Universal Robots PolyScope program: WIE2.urp

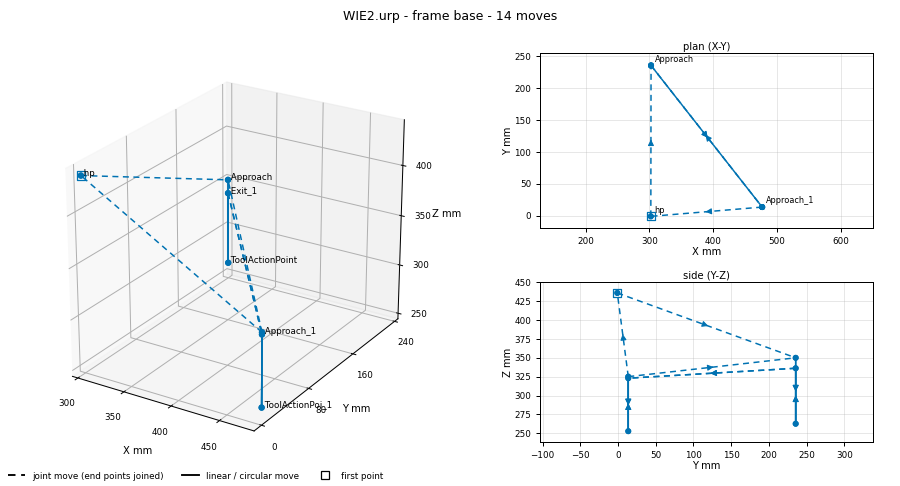
[picture p0: tool path of WIE2.urp in frame base, 14 of 14 moves have a stored position in this frame; points joined in program order, loops and branches not executed]
Program WIE2 (installation=default directory=/programs/Students createdIn=5.11.9.1010452 lastSavedIn=5.11.9.1010452 robotSerialNumber=20225200364)
Calibrated DH parameters: a=[0.00002, -0.569483, -0.54992, -0.00001, -0.000036, 0]; d=[0.180894, -146.691669, 192.918669, -46.053088, 0.119778, 0.115602]; alpha=[1.571425, -0.001534, 0.003359, 1.568739, -1.571477, 0]; deltaTheta=[0, 0.376258, -0.101074, -0.275185, -0.000002, 0]
Robot Program (runOnlyOnce=false)
  URCap RG Grip (OnRobot, OnRobot A/S) dataModel(rg-target-force=40.0, rg-target-width=0.1, Variable(key=on_return, variable(name=on_return)))
  MoveJ speed 60 deg/s, acceleration 80 deg/s^2 (useActiveTCP=true) feature=Base
    Waypoint hp: TCP in base x=302.217 y=-0.87 z=436.088 mm, rx=2.2254 ry=-2.21 rz=0.0041 rad; joints [35.141, -74.845, -127.965, -247.503, -90.009, -145.045] deg
    Loop Counting (count=3) loopVariable(name=Loop_1)
      URCap Palletizing (polyscope-pallet-impl, Universal Robots) dataModel(palletFeature=Base, isPalletizing=true, Variable(key=name, variable(name=Pallet_1)), Variable(key=globalCountingVariable, variable(name=Pallet_1_cnt_1, initializeExpression=1)), Variable(key=layerNumberVariable, variable(name=Pallet_1_lno, initializeExpression=1)), Variable(key=layerCountingVariable, variable(name=Pallet_1_lct, initializeExpression=1)), Variable(key=handleSeparatorVariable, variable(name=Pallet_1_sep, initializeExpression=False)), Variable(key=totalCountVariable, variable(name=Pallet_1_tct, initializeExpression=1)), Length(key=objectHeight value=0.00001 unit=M), Variable(key=referencePoint, variable(featureName=referencePoint)), Variable(key=separatorPoint, variable(featureName=separatorPoint))); state(isChildrenLocked=true)
        URCap Patterns (polyscope-pallet-impl, Universal Robots) state(isChildrenLocked=true)
          URCap Pattern (polyscope-pallet-impl, Universal Robots) dataModel(UUID=b11b03bd-8caf-4562-8920-b140e7a550b2, patternType=LINE, objects=3, Variable(key=nameVariable, variable(name=Line_Pattern_1))); state(isChildrenLocked=true)
            URCap Item (polyscope-pallet-impl, Universal Robots) dataModel(UUID=68741ad4-6990-4c8e-a16e-338bb588d268, patternType=LINE, index=0, calibrationDeltaTheta=[-2.1094217540068572E-7, 0.37625772532806073, -0.10107441100396769, -0.2751850025766889, -1.8024952768980196E-6, 2.9402326063437956E-8], calibrationA=[2.0416891277915125E-5, -0.5694828868469309, -0.5499202125525207, -9.504674691390763E-6, -3.603723657207661E-5, 0.0], calibrationD=[0.1808937726775539, -146.69166934821124, 192.91866861971778, -46.05308757405963, 0.11977780403821288, 0.11560212559305974], calibrationAlpha=[1.5714252480212174, -0.0015337665762078037, 0.0033588312559612306, 1.5687392298942362, -1.5714772428732047, 0.0], calibrationJointChecksum=[-1490546360, -1456574554, -1506622700, -1493399207, -1492840923, -1492940558], calibrationStatus=2, calibrationValidChecksum=true, baseToFeature=[0.0, 0.0, 0.0, 0.0, 0.0, 0.0], TCPOffset=[1.9606048756726224E-7, 3.440182682445947E-6, -6.058388327678799E-6, 3.4021623271823385E-5, 2.0407876993438444E-5, -5.7287062263560195E-5], Variable(key=variable, variable(name=StartItem_1)), JointPositions(key=jointpositions, JointPosition(key=[1], Angle(key=pos value=1.151144 unit=RAD)), JointPosition(key=[2], Angle(key=pos value=-1.665254 unit=RAD)), JointPosition(key=[3], Angle(key=pos value=-2.27469 unit=RAD)), JointPosition(key=[4], Angle(key=pos value=-3.920441 unit=RAD)), JointPosition(key=[5], Angle(key=pos value=-1.573051 unit=RAD)), JointPosition(key=[6], Angle(key=pos value=-1.992156 unit=RAD))))
            URCap Item (polyscope-pallet-impl, Universal Robots) dataModel(UUID=55b1d08e-faf5-4680-8923-1654362d1ff2, patternType=LINE, index=1, calibrationDeltaTheta=[-2.1094217540068572E-7, 0.37625772532806073, -0.10107441100396769, -0.2751850025766889, -1.8024952768980196E-6, 2.9402326063437956E-8], calibrationA=[2.0416891277915125E-5, -0.5694828868469309, -0.5499202125525207, -9.504674691390763E-6, -3.603723657207661E-5, 0.0], calibrationD=[0.1808937726775539, -146.69166934821124, 192.91866861971778, -46.05308757405963, 0.11977780403821288, 0.11560212559305974], calibrationAlpha=[1.5714252480212174, -0.0015337665762078037, 0.0033588312559612306, 1.5687392298942362, -1.5714772428732047, 0.0], calibrationJointChecksum=[-1490546360, -1456574554, -1506622700, -1493399207, -1492840923, -1492940558], calibrationStatus=2, calibrationValidChecksum=true, baseToFeature=[0.0, 0.0, 0.0, 0.0, 0.0, 0.0], TCPOffset=[1.6074322131992558E-5, 7.363046531760897E-6, 1.925072456621102E-5, 3.1824736687356776E-6, 3.869313491192138E-5, -4.1629896519852954E-5], Variable(key=variable, variable(name=EndItem_1)), JointPositions(key=jointpositions, JointPosition(key=[1], Angle(key=pos value=1.297803 unit=RAD)), JointPosition(key=[2], Angle(key=pos value=-1.600044 unit=RAD)), JointPosition(key=[3], Angle(key=pos value=-2.346172 unit=RAD)), JointPosition(key=[4], Angle(key=pos value=-3.914209 unit=RAD)), JointPosition(key=[5], Angle(key=pos value=-1.573925 unit=RAD)), JointPosition(key=[6], Angle(key=pos value=-1.845408 unit=RAD))))
        URCap Layers (polyscope-pallet-impl, Universal Robots) dataModel(separators=[false], selectedPatterns=[b11b03bd-8caf-4562-8920-b140e7a550b2])
        URCap At Each Item (polyscope-pallet-impl, Universal Robots) dataModel(selectedPattern=b11b03bd-8caf-4562-8920-b140e7a550b2, selectedPosition=68741ad4-6990-4c8e-a16e-338bb588d268, Approach_calibrationDeltaTheta=[-2.1094217540068572E-7, 0.37625772532806073, -0.10107441100396769, -0.2751850025766889, -1.8024952768980196E-6, 2.9402326063437956E-8], Approach_calibrationA=[2.0416891277915125E-5, -0.5694828868469309, -0.5499202125525207, -9.504674691390763E-6, -3.603723657207661E-5, 0.0], Approach_calibrationD=[0.1808937726775539, -146.69166934821124, 192.91866861971778, -46.05308757405963, 0.11977780403821288, 0.11560212559305974], Approach_calibrationAlpha=[1.5714252480212174, -0.0015337665762078037, 0.0033588312559612306, 1.5687392298942362, -1.5714772428732047, 0.0], Approach_calibrationJointChecksum=[-1490546360, -1456574554, -1506622700, -1493399207, -1492840923, -1492940558], Approach_calibrationStatus=2, Approach_calibrationValidChecksum=true, Approach_baseToFeature=[0.0, 0.0, 0.0, 0.0, 0.0, 0.0], Approach_TCPOffset=[-1.025128913775819E-5, 2.673478713677291E-5, 9.183253837474759E-6, -1.0917233999131985E-5, -2.1564629862661836E-5, -6.92566800690253E-5], Exit_calibrationDeltaTheta=[-2.1094217540068572E-7, 0.37625772532806073, -0.10107441100396769, -0.2751850025766889, -1.8024952768980196E-6, 2.9402326063437956E-8], Exit_calibrationA=[2.0416891277915125E-5, -0.5694828868469309, -0.5499202125525207, -9.504674691390763E-6, -3.603723657207661E-5, 0.0], Exit_calibrationD=[0.1808937726775539, -146.69166934821124, 192.91866861971778, -46.05308757405963, 0.11977780403821288, 0.11560212559305974], Exit_calibrationAlpha=[1.5714252480212174, -0.0015337665762078037, 0.0033588312559612306, 1.5687392298942362, -1.5714772428732047, 0.0], Exit_calibrationJointChecksum=[-1490546360, -1456574554, -1506622700, -1493399207, -1492840923, -1492940558], Exit_calibrationStatus=2, Exit_calibrationValidChecksum=true, Exit_baseToFeature=[0.0, 0.0, 0.0, 0.0, 0.0, 0.0], Exit_TCPOffset=[-1.3626013072698395E-5, 1.0862932783961554E-5, 1.1430969837411542E-5, -1.6285610609812615E-5, -7.832042440234011E-6, -7.245380913611749E-5], currentWizardState=SHOW_DONE, Pose(key=refBaseToFeature, Position(key=posePosition, Length(key=X value=0 unit=M), Length(key=Y value=0 unit=M), Length(key=Z value=0 unit=M)), Rotation(key=poseRotation, Angle(key=RX value=0 unit=RAD), Angle(key=RY value=0 unit=RAD), Angle(key=RZ value=0 unit=RAD))), Pose(key=refPose, Position(key=posePosition, Length(key=X value=0.302581 unit=M), Length(key=Y value=0.235564 unit=M), Length(key=Z value=0.265701 unit=M)), Rotation(key=poseRotation, Angle(key=RX value=2.225304 unit=RAD), Angle(key=RY value=-2.210079 unit=RAD), Angle(key=RZ value=0.003971 unit=RAD))), JointPositions(key=Approach_jointpositions, JointPosition(key=[1], Angle(key=pos value=1.133533 unit=RAD)), JointPosition(key=[2], Angle(key=pos value=-1.561307 unit=RAD)), JointPosition(key=[3], Angle(key=pos value=-2.193362 unit=RAD)), JointPosition(key=[4], Angle(key=pos value=-4.105764 unit=RAD)), JointPosition(key=[5], Angle(key=pos value=-1.57332 unit=RAD)), JointPosition(key=[6], Angle(key=pos value=-2.010341 unit=RAD))), JointPositions(key=Exit_jointpositions, JointPosition(key=[1], Angle(key=pos value=1.133574 unit=RAD)), JointPosition(key=[2], Angle(key=pos value=-1.577708 unit=RAD)), JointPosition(key=[3], Angle(key=pos value=-2.206947 unit=RAD)), JointPosition(key=[4], Angle(key=pos value=-4.075778 unit=RAD)), JointPosition(key=[5], Angle(key=pos value=-1.573263 unit=RAD)), JointPosition(key=[6], Angle(key=pos value=-2.010196 unit=RAD))))
          URCap Generated Movements (polyscope-pallet-impl, Universal Robots) state(isChildrenLocked=true)
            MoveJ speed 60 deg/s, acceleration 80 deg/s^2 (useActiveTCP=true) feature=referencePoint
              Waypoint Approach: TCP in base x=302.563 y=235.603 z=350.112 mm, rx=2.2254 ry=-2.2101 rz=0.0039 rad; joints [64.951, -89.455, -125.672, -235.241, -90.146, -115.184] deg; TCP offset x=0 y=0 z=0 mm, rx=0 ry=0 rz=0 rad; feature pose in base x=302.581 y=235.564 z=265.701 mm, rx=2.2253 ry=-2.2101 rz=0.004 rad
            MoveL speed 250 mm/s, acceleration 1200 mm/s^2 (useActiveTCP=true) feature(featureName=referencePoint)
              Waypoint ToolActionPoint: TCP in base x=302.59 y=235.593 z=262.688 mm, rx=2.2253 ry=-2.2101 rz=0.004 rad; joints [64.96, -96.193, -130.031, -224.145, -90.119, -115.133] deg; TCP offset x=0 y=0 z=0 mm, rx=0 ry=0 rz=0 rad
            Folder Tool action
              URCap RG Grip (OnRobot, OnRobot A/S) dataModel(rg-target-force=40.0, rg-target-width=0.075)
            MoveL speed 250 mm/s, acceleration 1200 mm/s^2 (useActiveTCP=true) feature(featureName=referencePoint)
              Waypoint Exit_1: TCP in base x=302.579 y=235.606 z=336.248 mm, rx=2.2254 ry=-2.21 rz=0.0039 rad; joints [64.951, -90.397, -126.449, -233.523, -90.142, -115.178] deg; TCP offset x=0 y=0 z=0 mm, rx=0 ry=0 rz=0 rad
      URCap Palletizing (polyscope-pallet-impl, Universal Robots) dataModel(palletFeature=Base, isPalletizing=true, Variable(key=name, variable(name=Pallet_2)), Variable(key=globalCountingVariable, variable(name=Pallet_2_cnt, initializeExpression=1)), Variable(key=layerNumberVariable, variable(name=Pallet_2_lno, initializeExpression=1)), Variable(key=layerCountingVariable, variable(name=Pallet_2_lct, initializeExpression=1)), Variable(key=handleSeparatorVariable, variable(name=Pallet_2_sep, initializeExpression=False)), Variable(key=totalCountVariable, variable(name=Pallet_2_tct, initializeExpression=1)), Variable(key=referencePoint, variable(featureName=referencePoin_1)), Variable(key=separatorPoint, variable(featureName=separatorPoin_1)), Length(key=objectHeight value=0.00001 unit=M)); state(isChildrenLocked=true)
        URCap Patterns (polyscope-pallet-impl, Universal Robots) state(isChildrenLocked=true)
          URCap Pattern (polyscope-pallet-impl, Universal Robots) dataModel(UUID=c499b9dd-d2c8-41fa-8b40-bf282c3e5683, patternType=LINE, objects=3, Variable(key=nameVariable, variable(name=Line_Pattern_2))); state(isChildrenLocked=true)
            URCap Item (polyscope-pallet-impl, Universal Robots) dataModel(UUID=52837b8f-e154-4d5d-bffa-9f20a0ef4224, patternType=LINE, index=0, calibrationDeltaTheta=[-2.1094217540068572E-7, 0.37625772532806073, -0.10107441100396769, -0.2751850025766889, -1.8024952768980196E-6, 2.9402326063437956E-8], calibrationA=[2.0416891277915125E-5, -0.5694828868469309, -0.5499202125525207, -9.504674691390763E-6, -3.603723657207661E-5, 0.0], calibrationD=[0.1808937726775539, -146.69166934821124, 192.91866861971778, -46.05308757405963, 0.11977780403821288, 0.11560212559305974], calibrationAlpha=[1.5714252480212174, -0.0015337665762078037, 0.0033588312559612306, 1.5687392298942362, -1.5714772428732047, 0.0], calibrationJointChecksum=[-1490546360, -1456574554, -1506622700, -1493399207, -1492840923, -1492940558], calibrationStatus=2, calibrationValidChecksum=true, baseToFeature=[0.0, 0.0, 0.0, 0.0, 0.0, 0.0], TCPOffset=[-2.1539357017180683E-5, -2.4505586607270757E-5, -2.766211884108749E-6, 1.7255755197503596E-5, 2.5774896433158367E-5, -3.127859189544208E-5], Variable(key=variable, variable(name=StartItem_2)), JointPositions(key=jointpositions, JointPosition(key=[1], Angle(key=pos value=0.404507 unit=RAD)), JointPosition(key=[2], Angle(key=pos value=-1.808746 unit=RAD)), JointPosition(key=[3], Angle(key=pos value=-2.094452 unit=RAD)), JointPosition(key=[4], Angle(key=pos value=-3.949963 unit=RAD)), JointPosition(key=[5], Angle(key=pos value=-1.569047 unit=RAD)), JointPosition(key=[6], Angle(key=pos value=-2.738939 unit=RAD))))
            URCap Item (polyscope-pallet-impl, Universal Robots) dataModel(UUID=17c72c05-39d8-4f72-8957-83a1ae3738ac, patternType=LINE, index=1, calibrationDeltaTheta=[-2.1094217540068572E-7, 0.37625772532806073, -0.10107441100396769, -0.2751850025766889, -1.8024952768980196E-6, 2.9402326063437956E-8], calibrationA=[2.0416891277915125E-5, -0.5694828868469309, -0.5499202125525207, -9.504674691390763E-6, -3.603723657207661E-5, 0.0], calibrationD=[0.1808937726775539, -146.69166934821124, 192.91866861971778, -46.05308757405963, 0.11977780403821288, 0.11560212559305974], calibrationAlpha=[1.5714252480212174, -0.0015337665762078037, 0.0033588312559612306, 1.5687392298942362, -1.5714772428732047, 0.0], calibrationJointChecksum=[-1490546360, -1456574554, -1506622700, -1493399207, -1492840923, -1492940558], calibrationStatus=2, calibrationValidChecksum=true, baseToFeature=[0.0, 0.0, 0.0, 0.0, 0.0, 0.0], TCPOffset=[-8.331917916487921E-6, -3.211176514195113E-6, -1.917540110196736E-5, 1.7094779368867274E-5, -3.4621062932593835E-5, -1.99212577807049E-5], Variable(key=variable, variable(name=EndItem_2)), JointPositions(key=jointpositions, JointPosition(key=[1], Angle(key=pos value=0.456202 unit=RAD)), JointPosition(key=[2], Angle(key=pos value=-1.732026 unit=RAD)), JointPosition(key=[3], Angle(key=pos value=-2.194038 unit=RAD)), JointPosition(key=[4], Angle(key=pos value=-3.927322 unit=RAD)), JointPosition(key=[5], Angle(key=pos value=-1.569054 unit=RAD)), JointPosition(key=[6], Angle(key=pos value=-2.687197 unit=RAD))))
        URCap Layers (polyscope-pallet-impl, Universal Robots) dataModel(separators=[false], selectedPatterns=[c499b9dd-d2c8-41fa-8b40-bf282c3e5683])
        URCap At Each Item (polyscope-pallet-impl, Universal Robots) dataModel(selectedPattern=c499b9dd-d2c8-41fa-8b40-bf282c3e5683, selectedPosition=52837b8f-e154-4d5d-bffa-9f20a0ef4224, Approach_calibrationDeltaTheta=[-2.1094217540068572E-7, 0.37625772532806073, -0.10107441100396769, -0.2751850025766889, -1.8024952768980196E-6, 2.9402326063437956E-8], Approach_calibrationA=[2.0416891277915125E-5, -0.5694828868469309, -0.5499202125525207, -9.504674691390763E-6, -3.603723657207661E-5, 0.0], Approach_calibrationD=[0.1808937726775539, -146.69166934821124, 192.91866861971778, -46.05308757405963, 0.11977780403821288, 0.11560212559305974], Approach_calibrationAlpha=[1.5714252480212174, -0.0015337665762078037, 0.0033588312559612306, 1.5687392298942362, -1.5714772428732047, 0.0], Approach_calibrationJointChecksum=[-1490546360, -1456574554, -1506622700, -1493399207, -1492840923, -1492940558], Approach_calibrationStatus=2, Approach_calibrationValidChecksum=true, Approach_baseToFeature=[0.0, 0.0, 0.0, 0.0, 0.0, 0.0], Approach_TCPOffset=[-9.24481925559939E-6, -4.320892813325372E-6, 3.208681495281418E-6, 1.5618489079231655E-5, 4.887824156400097E-6, 3.115654338511915E-6], Exit_calibrationDeltaTheta=[-2.1094217540068572E-7, 0.37625772532806073, -0.10107441100396769, -0.2751850025766889, -1.8024952768980196E-6, 2.9402326063437956E-8], Exit_calibrationA=[2.0416891277915125E-5, -0.5694828868469309, -0.5499202125525207, -9.504674691390763E-6, -3.603723657207661E-5, 0.0], Exit_calibrationD=[0.1808937726775539, -146.69166934821124, 192.91866861971778, -46.05308757405963, 0.11977780403821288, 0.11560212559305974], Exit_calibrationAlpha=[1.5714252480212174, -0.0015337665762078037, 0.0033588312559612306, 1.5687392298942362, -1.5714772428732047, 0.0], Exit_calibrationJointChecksum=[-1490546360, -1456574554, -1506622700, -1493399207, -1492840923, -1492940558], Exit_calibrationStatus=2, Exit_calibrationValidChecksum=true, Exit_baseToFeature=[0.0, 0.0, 0.0, 0.0, 0.0, 0.0], Exit_TCPOffset=[-5.158242497903601E-6, -3.725374339402787E-6, 1.8701733796033793E-5, -4.294771303553589E-5, 2.7081890225548673E-5, 7.0994869539825734E-6], currentWizardState=SHOW_DONE, Pose(key=refBaseToFeature, Position(key=posePosition, Length(key=X value=0 unit=M), Length(key=Y value=0 unit=M), Length(key=Z value=0 unit=M)), Rotation(key=poseRotation, Angle(key=RX value=0 unit=RAD), Angle(key=RY value=0 unit=RAD), Angle(key=RZ value=0 unit=RAD))), Pose(key=refPose, Position(key=posePosition, Length(key=X value=0.476779 unit=M), Length(key=Y value=0.013666 unit=M), Length(key=Z value=0.252817 unit=M)), Rotation(key=poseRotation, Angle(key=RX value=2.225541 unit=RAD), Angle(key=RY value=-2.210024 unit=RAD), Angle(key=RZ value=0.003865 unit=RAD))), JointPositions(key=Approach_jointpositions, JointPosition(key=[1], Angle(key=pos value=0.403596 unit=RAD)), JointPosition(key=[2], Angle(key=pos value=-1.749254 unit=RAD)), JointPosition(key=[3], Angle(key=pos value=-2.04242 unit=RAD)), JointPosition(key=[4], Angle(key=pos value=-4.06685 unit=RAD)), JointPosition(key=[5], Angle(key=pos value=-1.569381 unit=RAD)), JointPosition(key=[6], Angle(key=pos value=-2.740204 unit=RAD))), JointPositions(key=Exit_jointpositions, JointPosition(key=[1], Angle(key=pos value=0.403593 unit=RAD)), JointPosition(key=[2], Angle(key=pos value=-1.746959 unit=RAD)), JointPosition(key=[3], Angle(key=pos value=-2.040696 unit=RAD)), JointPosition(key=[4], Angle(key=pos value=-4.070868 unit=RAD)), JointPosition(key=[5], Angle(key=pos value=-1.569389 unit=RAD)), JointPosition(key=[6], Angle(key=pos value=-2.740221 unit=RAD))))
          URCap Generated Movements (polyscope-pallet-impl, Universal Robots) state(isChildrenLocked=true)
            MoveJ speed 60 deg/s, acceleration 80 deg/s^2 (useActiveTCP=true) feature=referencePoin_1
              Waypoint Approach_1: TCP in base x=476.783 y=13.675 z=323.071 mm, rx=2.2255 ry=-2.21 rz=0.0039 rad; joints [23.125, -100.225, -117.022, -233.012, -89.918, -157.001] deg; TCP offset x=0 y=0 z=0 mm, rx=0 ry=0 rz=0 rad; feature pose in base x=476.779 y=13.666 z=252.817 mm, rx=2.2255 ry=-2.21 rz=0.0039 rad
            MoveL speed 250 mm/s, acceleration 1200 mm/s^2 (useActiveTCP=true) feature(featureName=referencePoin_1)
              Waypoint ToolActionPoi_1: TCP in base x=476.779 y=13.666 z=252.817 mm, rx=2.2255 ry=-2.21 rz=0.0039 rad; joints [23.13, -105.137, -119.931, -225.193, -89.9, -156.972] deg; TCP offset x=0 y=0 z=0 mm, rx=0 ry=0 rz=0 rad
            Folder Tool action
              URCap RG Grip (OnRobot, OnRobot A/S) dataModel(rg-target-force=40.0, rg-target-width=0.1)
            MoveL speed 250 mm/s, acceleration 1200 mm/s^2 (useActiveTCP=true) feature(featureName=referencePoin_1)
              Waypoint Exit_2: TCP in base x=476.782 y=13.671 z=325.136 mm, rx=2.2255 ry=-2.21 rz=0.0038 rad; joints [23.125, -100.096, -116.923, -233.244, -89.919, -157.002] deg; TCP offset x=0 y=0 z=0 mm, rx=0 ry=0 rz=0 rad
    Loop Counting (count=3) loopVariable(name=Loop_2)
      URCap Palletizing (polyscope-pallet-impl, Universal Robots) dataModel(palletFeature=Base, isPalletizing=true, Length(key=objectHeight value=0.00001 unit=M), Variable(key=name, variable(name=Pallet_3)), Variable(key=globalCountingVariable, variable(name=Pallet_3_cnt, initializeExpression=1)), Variable(key=layerNumberVariable, variable(name=Pallet_3_lno, initializeExpression=1)), Variable(key=layerCountingVariable, variable(name=Pallet_3_lct, initializeExpression=1)), Variable(key=handleSeparatorVariable, variable(name=Pallet_3_sep, initializeExpression=False)), Variable(key=totalCountVariable, variable(name=Pallet_3_tct, initializeExpression=1)), Variable(key=referencePoint, variable(featureName=referencePoin_2)), Variable(key=separatorPoint, variable(featureName=separatorPoin_2))); state(isChildrenLocked=true)
        URCap Patterns (polyscope-pallet-impl, Universal Robots) state(isChildrenLocked=true)
          URCap Pattern (polyscope-pallet-impl, Universal Robots) dataModel(UUID=b11b03bd-8caf-4562-8920-b140e7a550b2, patternType=LINE, objects=3, Variable(key=nameVariable, variable(name=Line_Pattern_3))); state(isChildrenLocked=true)
            URCap Item (polyscope-pallet-impl, Universal Robots) dataModel(UUID=68741ad4-6990-4c8e-a16e-338bb588d268, patternType=LINE, index=0, calibrationDeltaTheta=[-2.1094217540068572E-7, 0.37625772532806073, -0.10107441100396769, -0.2751850025766889, -1.8024952768980196E-6, 2.9402326063437956E-8], calibrationA=[2.0416891277915125E-5, -0.5694828868469309, -0.5499202125525207, -9.504674691390763E-6, -3.603723657207661E-5, 0.0], calibrationD=[0.1808937726775539, -146.69166934821124, 192.91866861971778, -46.05308757405963, 0.11977780403821288, 0.11560212559305974], calibrationAlpha=[1.5714252480212174, -0.0015337665762078037, 0.0033588312559612306, 1.5687392298942362, -1.5714772428732047, 0.0], calibrationJointChecksum=[-1490546360, -1456574554, -1506622700, -1493399207, -1492840923, -1492940558], calibrationStatus=2, calibrationValidChecksum=true, baseToFeature=[0.0, 0.0, 0.0, 0.0, 0.0, 0.0], TCPOffset=[-3.1843261568687E-6, -1.1922170369549345E-6, 5.402865667081258E-7, -1.7557571740777845E-5, 6.471469548214763E-6, 5.889117264410654E-6], Variable(key=variable, variable(name=StartItem_3)), JointPositions(key=jointpositions, JointPosition(key=[1], Angle(key=pos value=1.383133 unit=RAD)), JointPosition(key=[2], Angle(key=pos value=-1.566893 unit=RAD)), JointPosition(key=[3], Angle(key=pos value=-2.379939 unit=RAD)), JointPosition(key=[4], Angle(key=pos value=-3.913497 unit=RAD)), JointPosition(key=[5], Angle(key=pos value=-1.574533 unit=RAD)), JointPosition(key=[6], Angle(key=pos value=-1.760152 unit=RAD))))
            URCap Item (polyscope-pallet-impl, Universal Robots) dataModel(UUID=55b1d08e-faf5-4680-8923-1654362d1ff2, patternType=LINE, index=1, calibrationDeltaTheta=[-2.1094217540068572E-7, 0.37625772532806073, -0.10107441100396769, -0.2751850025766889, -1.8024952768980196E-6, 2.9402326063437956E-8], calibrationA=[2.0416891277915125E-5, -0.5694828868469309, -0.5499202125525207, -9.504674691390763E-6, -3.603723657207661E-5, 0.0], calibrationD=[0.1808937726775539, -146.69166934821124, 192.91866861971778, -46.05308757405963, 0.11977780403821288, 0.11560212559305974], calibrationAlpha=[1.5714252480212174, -0.0015337665762078037, 0.0033588312559612306, 1.5687392298942362, -1.5714772428732047, 0.0], calibrationJointChecksum=[-1490546360, -1456574554, -1506622700, -1493399207, -1492840923, -1492940558], calibrationStatus=2, calibrationValidChecksum=true, baseToFeature=[0.0, 0.0, 0.0, 0.0, 0.0, 0.0], TCPOffset=[3.3905110172205433E-6, -1.3686699736892294E-6, -2.00069086438992E-5, -7.064266040329533E-6, -1.5420028567504033E-5, 1.3232124956267159E-5], Variable(key=variable, variable(name=EndItem_3)), JointPositions(key=jointpositions, JointPosition(key=[1], Angle(key=pos value=1.573984 unit=RAD)), JointPosition(key=[2], Angle(key=pos value=-1.502491 unit=RAD)), JointPosition(key=[3], Angle(key=pos value=-2.440712 unit=RAD)), JointPosition(key=[4], Angle(key=pos value=-3.916849 unit=RAD)), JointPosition(key=[5], Angle(key=pos value=-1.57569 unit=RAD)), JointPosition(key=[6], Angle(key=pos value=-1.569354 unit=RAD))))
        URCap Layers (polyscope-pallet-impl, Universal Robots) dataModel(separators=[false], selectedPatterns=[b11b03bd-8caf-4562-8920-b140e7a550b2])
        URCap At Each Item (polyscope-pallet-impl, Universal Robots) dataModel(selectedPattern=b11b03bd-8caf-4562-8920-b140e7a550b2, selectedPosition=68741ad4-6990-4c8e-a16e-338bb588d268, Approach_calibrationDeltaTheta=[-2.1094217540068572E-7, 0.37625772532806073, -0.10107441100396769, -0.2751850025766889, -1.8024952768980196E-6, 2.9402326063437956E-8], Approach_calibrationA=[2.0416891277915125E-5, -0.5694828868469309, -0.5499202125525207, -9.504674691390763E-6, -3.603723657207661E-5, 0.0], Approach_calibrationD=[0.1808937726775539, -146.69166934821124, 192.91866861971778, -46.05308757405963, 0.11977780403821288, 0.11560212559305974], Approach_calibrationAlpha=[1.5714252480212174, -0.0015337665762078037, 0.0033588312559612306, 1.5687392298942362, -1.5714772428732047, 0.0], Approach_calibrationJointChecksum=[-1490546360, -1456574554, -1506622700, -1493399207, -1492840923, -1492940558], Approach_calibrationStatus=2, Approach_calibrationValidChecksum=true, Approach_baseToFeature=[0.0, 0.0, 0.0, 0.0, 0.0, 0.0], Approach_TCPOffset=[-1.025128913775819E-5, 2.673478713677291E-5, 9.183253837474759E-6, -1.0917233999131985E-5, -2.1564629862661836E-5, -6.92566800690253E-5], Exit_calibrationDeltaTheta=[-2.1094217540068572E-7, 0.37625772532806073, -0.10107441100396769, -0.2751850025766889, -1.8024952768980196E-6, 2.9402326063437956E-8], Exit_calibrationA=[2.0416891277915125E-5, -0.5694828868469309, -0.5499202125525207, -9.504674691390763E-6, -3.603723657207661E-5, 0.0], Exit_calibrationD=[0.1808937726775539, -146.69166934821124, 192.91866861971778, -46.05308757405963, 0.11977780403821288, 0.11560212559305974], Exit_calibrationAlpha=[1.5714252480212174, -0.0015337665762078037, 0.0033588312559612306, 1.5687392298942362, -1.5714772428732047, 0.0], Exit_calibrationJointChecksum=[-1490546360, -1456574554, -1506622700, -1493399207, -1492840923, -1492940558], Exit_calibrationStatus=2, Exit_calibrationValidChecksum=true, Exit_baseToFeature=[0.0, 0.0, 0.0, 0.0, 0.0, 0.0], Exit_TCPOffset=[-1.3626013072698395E-5, 1.0862932783961554E-5, 1.1430969837411542E-5, -1.6285610609812615E-5, -7.832042440234011E-6, -7.245380913611749E-5], currentWizardState=SHOW_DONE, Pose(key=refBaseToFeature, Position(key=posePosition, Length(key=X value=0 unit=M), Length(key=Y value=0 unit=M), Length(key=Z value=0 unit=M)), Rotation(key=poseRotation, Angle(key=RX value=0 unit=RAD), Angle(key=RY value=0 unit=RAD), Angle(key=RZ value=0 unit=RAD))), Pose(key=refPose, Position(key=posePosition, Length(key=X value=0.302581 unit=M), Length(key=Y value=0.235564 unit=M), Length(key=Z value=0.265701 unit=M)), Rotation(key=poseRotation, Angle(key=RX value=2.225304 unit=RAD), Angle(key=RY value=-2.210079 unit=RAD), Angle(key=RZ value=0.003971 unit=RAD))), JointPositions(key=Approach_jointpositions, JointPosition(key=[1], Angle(key=pos value=1.133533 unit=RAD)), JointPosition(key=[2], Angle(key=pos value=-1.561307 unit=RAD)), JointPosition(key=[3], Angle(key=pos value=-2.193362 unit=RAD)), JointPosition(key=[4], Angle(key=pos value=-4.105764 unit=RAD)), JointPosition(key=[5], Angle(key=pos value=-1.57332 unit=RAD)), JointPosition(key=[6], Angle(key=pos value=-2.010341 unit=RAD))), JointPositions(key=Exit_jointpositions, JointPosition(key=[1], Angle(key=pos value=1.133574 unit=RAD)), JointPosition(key=[2], Angle(key=pos value=-1.577708 unit=RAD)), JointPosition(key=[3], Angle(key=pos value=-2.206947 unit=RAD)), JointPosition(key=[4], Angle(key=pos value=-4.075778 unit=RAD)), JointPosition(key=[5], Angle(key=pos value=-1.573263 unit=RAD)), JointPosition(key=[6], Angle(key=pos value=-2.010196 unit=RAD))))
          URCap Generated Movements (polyscope-pallet-impl, Universal Robots) state(isChildrenLocked=true)
            MoveJ speed 60 deg/s, acceleration 80 deg/s^2 (useActiveTCP=true) feature=referencePoin_2
              Waypoint Approach: TCP in base x=302.563 y=235.603 z=350.112 mm, rx=2.2254 ry=-2.2101 rz=0.0039 rad; joints [64.951, -89.455, -125.672, -235.241, -90.146, -115.184] deg; TCP offset x=0 y=0 z=0 mm, rx=0 ry=0 rz=0 rad; feature pose in base x=302.581 y=235.564 z=265.701 mm, rx=2.2253 ry=-2.2101 rz=0.004 rad
            MoveL speed 250 mm/s, acceleration 1200 mm/s^2 (useActiveTCP=true) feature(featureName=referencePoin_2)
              Waypoint ToolActionPoint: TCP in base x=302.59 y=235.593 z=262.688 mm, rx=2.2253 ry=-2.2101 rz=0.004 rad; joints [64.96, -96.193, -130.031, -224.145, -90.119, -115.133] deg; TCP offset x=0 y=0 z=0 mm, rx=0 ry=0 rz=0 rad
            Folder Tool action
              URCap RG Grip (OnRobot, OnRobot A/S) dataModel(rg-target-force=40.0, rg-target-width=0.075)
            MoveL speed 250 mm/s, acceleration 1200 mm/s^2 (useActiveTCP=true) feature(featureName=referencePoin_2)
              Waypoint Exit_1: TCP in base x=302.579 y=235.606 z=336.248 mm, rx=2.2254 ry=-2.21 rz=0.0039 rad; joints [64.951, -90.397, -126.449, -233.523, -90.142, -115.178] deg; TCP offset x=0 y=0 z=0 mm, rx=0 ry=0 rz=0 rad
      URCap Palletizing (polyscope-pallet-impl, Universal Robots) dataModel(palletFeature=Base, isPalletizing=true, Length(key=objectHeight value=0.00001 unit=M), Variable(key=name, variable(name=Pallet_4)), Variable(key=globalCountingVariable, variable(name=Pallet_4_cnt, initializeExpression=1)), Variable(key=layerNumberVariable, variable(name=Pallet_4_lno, initializeExpression=1)), Variable(key=layerCountingVariable, variable(name=Pallet_4_lct, initializeExpression=1)), Variable(key=handleSeparatorVariable, variable(name=Pallet_4_sep, initializeExpression=False)), Variable(key=totalCountVariable, variable(name=Pallet_4_tct, initializeExpression=1)), Variable(key=referencePoint, variable(featureName=referencePoin_3)), Variable(key=separatorPoint, variable(featureName=separatorPoin_3))); state(isChildrenLocked=true)
        URCap Patterns (polyscope-pallet-impl, Universal Robots) state(isChildrenLocked=true)
          URCap Pattern (polyscope-pallet-impl, Universal Robots) dataModel(UUID=c499b9dd-d2c8-41fa-8b40-bf282c3e5683, patternType=LINE, objects=3, Variable(key=nameVariable, variable(name=Line_Pattern_4))); state(isChildrenLocked=true)
            URCap Item (polyscope-pallet-impl, Universal Robots) dataModel(UUID=52837b8f-e154-4d5d-bffa-9f20a0ef4224, patternType=LINE, index=0, calibrationDeltaTheta=[-2.1094217540068572E-7, 0.37625772532806073, -0.10107441100396769, -0.2751850025766889, -1.8024952768980196E-6, 2.9402326063437956E-8], calibrationA=[2.0416891277915125E-5, -0.5694828868469309, -0.5499202125525207, -9.504674691390763E-6, -3.603723657207661E-5, 0.0], calibrationD=[0.1808937726775539, -146.69166934821124, 192.91866861971778, -46.05308757405963, 0.11977780403821288, 0.11560212559305974], calibrationAlpha=[1.5714252480212174, -0.0015337665762078037, 0.0033588312559612306, 1.5687392298942362, -1.5714772428732047, 0.0], calibrationJointChecksum=[-1490546360, -1456574554, -1506622700, -1493399207, -1492840923, -1492940558], calibrationStatus=2, calibrationValidChecksum=true, baseToFeature=[0.0, 0.0, 0.0, 0.0, 0.0, 0.0], TCPOffset=[1.3413943985129961E-5, 3.081082408285321E-5, -1.1130057322339404E-5, -1.744567229757518E-4, 7.096992480329918E-5, -7.137860935328706E-5], Variable(key=variable, variable(name=StartItem_4)), JointPositions(key=jointpositions, JointPosition(key=[1], Angle(key=pos value=0.364325 unit=RAD)), JointPosition(key=[2], Angle(key=pos value=-1.757491 unit=RAD)), JointPosition(key=[3], Angle(key=pos value=-2.125527 unit=RAD)), JointPosition(key=[4], Angle(key=pos value=-3.97598 unit=RAD)), JointPosition(key=[5], Angle(key=pos value=-1.571677 unit=RAD)), JointPosition(key=[6], Angle(key=pos value=-1.21622 unit=RAD))))
            URCap Item (polyscope-pallet-impl, Universal Robots) dataModel(UUID=17c72c05-39d8-4f72-8957-83a1ae3738ac, patternType=LINE, index=1, calibrationDeltaTheta=[-2.1094217540068572E-7, 0.37625772532806073, -0.10107441100396769, -0.2751850025766889, -1.8024952768980196E-6, 2.9402326063437956E-8], calibrationA=[2.0416891277915125E-5, -0.5694828868469309, -0.5499202125525207, -9.504674691390763E-6, -3.603723657207661E-5, 0.0], calibrationD=[0.1808937726775539, -146.69166934821124, 192.91866861971778, -46.05308757405963, 0.11977780403821288, 0.11560212559305974], calibrationAlpha=[1.5714252480212174, -0.0015337665762078037, 0.0033588312559612306, 1.5687392298942362, -1.5714772428732047, 0.0], calibrationJointChecksum=[-1490546360, -1456574554, -1506622700, -1493399207, -1492840923, -1492940558], calibrationStatus=2, calibrationValidChecksum=true, baseToFeature=[0.0, 0.0, 0.0, 0.0, 0.0, 0.0], TCPOffset=[-7.044407026590704E-6, -5.194365089632169E-6, -1.55428668031643E-5, 2.8640682100730482E-5, -2.286772933350867E-5, 1.38487609951116E-5], Variable(key=variable, variable(name=EndItem_4)), JointPositions(key=jointpositions, JointPosition(key=[1], Angle(key=pos value=0.472854 unit=RAD)), JointPosition(key=[2], Angle(key=pos value=-1.759448 unit=RAD)), JointPosition(key=[3], Angle(key=pos value=-2.123483 unit=RAD)), JointPosition(key=[4], Angle(key=pos value=-3.974312 unit=RAD)), JointPosition(key=[5], Angle(key=pos value=-1.575595 unit=RAD)), JointPosition(key=[6], Angle(key=pos value=-1.107685 unit=RAD))))
        URCap Layers (polyscope-pallet-impl, Universal Robots) dataModel(separators=[false], selectedPatterns=[c499b9dd-d2c8-41fa-8b40-bf282c3e5683])
        URCap At Each Item (polyscope-pallet-impl, Universal Robots) dataModel(selectedPattern=c499b9dd-d2c8-41fa-8b40-bf282c3e5683, selectedPosition=52837b8f-e154-4d5d-bffa-9f20a0ef4224, Approach_calibrationDeltaTheta=[-2.1094217540068572E-7, 0.37625772532806073, -0.10107441100396769, -0.2751850025766889, -1.8024952768980196E-6, 2.9402326063437956E-8], Approach_calibrationA=[2.0416891277915125E-5, -0.5694828868469309, -0.5499202125525207, -9.504674691390763E-6, -3.603723657207661E-5, 0.0], Approach_calibrationD=[0.1808937726775539, -146.69166934821124, 192.91866861971778, -46.05308757405963, 0.11977780403821288, 0.11560212559305974], Approach_calibrationAlpha=[1.5714252480212174, -0.0015337665762078037, 0.0033588312559612306, 1.5687392298942362, -1.5714772428732047, 0.0], Approach_calibrationJointChecksum=[-1490546360, -1456574554, -1506622700, -1493399207, -1492840923, -1492940558], Approach_calibrationStatus=2, Approach_calibrationValidChecksum=true, Approach_baseToFeature=[0.0, 0.0, 0.0, 0.0, 0.0, 0.0], Approach_TCPOffset=[-9.24481925559939E-6, -4.320892813325372E-6, 3.208681495281418E-6, 1.5618489079231655E-5, 4.887824156400097E-6, 3.115654338511915E-6], Exit_calibrationDeltaTheta=[-2.1094217540068572E-7, 0.37625772532806073, -0.10107441100396769, -0.2751850025766889, -1.8024952768980196E-6, 2.9402326063437956E-8], Exit_calibrationA=[2.0416891277915125E-5, -0.5694828868469309, -0.5499202125525207, -9.504674691390763E-6, -3.603723657207661E-5, 0.0], Exit_calibrationD=[0.1808937726775539, -146.69166934821124, 192.91866861971778, -46.05308757405963, 0.11977780403821288, 0.11560212559305974], Exit_calibrationAlpha=[1.5714252480212174, -0.0015337665762078037, 0.0033588312559612306, 1.5687392298942362, -1.5714772428732047, 0.0], Exit_calibrationJointChecksum=[-1490546360, -1456574554, -1506622700, -1493399207, -1492840923, -1492940558], Exit_calibrationStatus=2, Exit_calibrationValidChecksum=true, Exit_baseToFeature=[0.0, 0.0, 0.0, 0.0, 0.0, 0.0], Exit_TCPOffset=[-5.158242497903601E-6, -3.725374339402787E-6, 1.8701733796033793E-5, -4.294771303553589E-5, 2.7081890225548673E-5, 7.0994869539825734E-6], currentWizardState=SHOW_DONE, Pose(key=refBaseToFeature, Position(key=posePosition, Length(key=X value=0 unit=M), Length(key=Y value=0 unit=M), Length(key=Z value=0 unit=M)), Rotation(key=poseRotation, Angle(key=RX value=0 unit=RAD), Angle(key=RY value=0 unit=RAD), Angle(key=RZ value=0 unit=RAD))), Pose(key=refPose, Position(key=posePosition, Length(key=X value=0.476779 unit=M), Length(key=Y value=0.013666 unit=M), Length(key=Z value=0.252817 unit=M)), Rotation(key=poseRotation, Angle(key=RX value=2.225541 unit=RAD), Angle(key=RY value=-2.210024 unit=RAD), Angle(key=RZ value=0.003865 unit=RAD))), JointPositions(key=Approach_jointpositions, JointPosition(key=[1], Angle(key=pos value=0.403596 unit=RAD)), JointPosition(key=[2], Angle(key=pos value=-1.749254 unit=RAD)), JointPosition(key=[3], Angle(key=pos value=-2.04242 unit=RAD)), JointPosition(key=[4], Angle(key=pos value=-4.06685 unit=RAD)), JointPosition(key=[5], Angle(key=pos value=-1.569381 unit=RAD)), JointPosition(key=[6], Angle(key=pos value=-2.740204 unit=RAD))), JointPositions(key=Exit_jointpositions, JointPosition(key=[1], Angle(key=pos value=0.403593 unit=RAD)), JointPosition(key=[2], Angle(key=pos value=-1.746959 unit=RAD)), JointPosition(key=[3], Angle(key=pos value=-2.040696 unit=RAD)), JointPosition(key=[4], Angle(key=pos value=-4.070868 unit=RAD)), JointPosition(key=[5], Angle(key=pos value=-1.569389 unit=RAD)), JointPosition(key=[6], Angle(key=pos value=-2.740221 unit=RAD))))
          URCap Generated Movements (polyscope-pallet-impl, Universal Robots) state(isChildrenLocked=true)
            MoveJ speed 60 deg/s, acceleration 80 deg/s^2 (useActiveTCP=true) feature=referencePoin_3
              Waypoint Approach_1: TCP in base x=476.783 y=13.675 z=323.071 mm, rx=2.2255 ry=-2.21 rz=0.0039 rad; joints [23.125, -100.225, -117.022, -233.012, -89.918, -157.001] deg; TCP offset x=0 y=0 z=0 mm, rx=0 ry=0 rz=0 rad; feature pose in base x=476.779 y=13.666 z=252.817 mm, rx=2.2255 ry=-2.21 rz=0.0039 rad
            MoveL speed 250 mm/s, acceleration 1200 mm/s^2 (useActiveTCP=true) feature(featureName=referencePoin_3)
              Waypoint ToolActionPoi_1: TCP in base x=476.779 y=13.666 z=252.817 mm, rx=2.2255 ry=-2.21 rz=0.0039 rad; joints [23.13, -105.137, -119.931, -225.193, -89.9, -156.972] deg; TCP offset x=0 y=0 z=0 mm, rx=0 ry=0 rz=0 rad
            Folder Tool action
              URCap RG Grip (OnRobot, OnRobot A/S) dataModel(rg-target-force=40.0, rg-target-width=0.1)
            MoveL speed 250 mm/s, acceleration 1200 mm/s^2 (useActiveTCP=true) feature(featureName=referencePoin_3)
              Waypoint Exit_2: TCP in base x=476.782 y=13.671 z=325.136 mm, rx=2.2255 ry=-2.21 rz=0.0038 rad; joints [23.125, -100.096, -116.923, -233.244, -89.919, -157.002] deg; TCP offset x=0 y=0 z=0 mm, rx=0 ry=0 rz=0 rad
    Waypoint hp: TCP in base x=302.217 y=-0.87 z=436.088 mm, rx=2.2254 ry=-2.21 rz=0.0041 rad; joints [35.141, -74.845, -127.965, -247.503, -90.009, -145.045] deg
    Halt
